TYPE ST_Motor :
STRUCT
	fSpeedMax : REAL;
	fSpeedMin : REAL;
END_STRUCT
END_TYPE

(* stored: Version 1.1.0.1, ProductVersion 3.1.4024.12
   DUT ST_Motor: Id {49e9c45d-c525-4653-a0a5-a7ee3dc05834} *)
